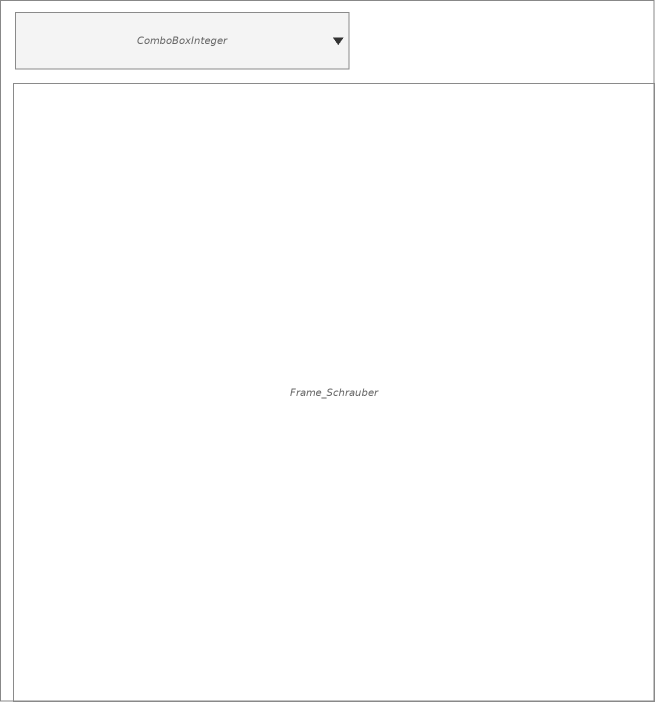
VISUALIZATION Schrauber_Aufruf  // 655x702
    Frame (13,83 642x619)
        shows Frame_Schrauber(stSKSSchrauberInOut := stSKSSchrauberInOut_Vis_Schr_1)
    ComboBoxInteger (15,12 334x57), variable: PRG_Schrauber.iAuswSchrauberMode, text list: 'TL_AuswahlSchrauberAblauf'
END_VISUALIZATION

(* stored: Version 1.1.0.1, ProductVersion 3.1.4024.15
   Visu Schrauber_Aufruf: Id {89c504c4-06fd-42fd-b8a7-8d0e4e4178aa} *)
